Staubli VAL3: regular_pick.pgx

program regular_pick(tool x_tTool, mdesc x_mMdesc, mdesc x_mMdesc_slow, point x_pPoint_pick, dio x_dDio_cy, bool x_bBool_bk, dio x_dDio_secure)
  local point l_pPoint_pick
  local point l_pPoint_safe
  local point l_pPoint_aprch
begin

  //vertical regular pick process

  //control point preparation
  l_pPoint_safe=x_pPoint_pick
  l_pPoint_safe.trsf.z=l_pPoint_safe.trsf.z+nNum_safe_h
  //approach point preparation
  l_pPoint_aprch=x_pPoint_pick
  l_pPoint_aprch.trsf.z=l_pPoint_aprch.trsf.z+nNum_apporach_h
  //pick point preparation
  l_pPoint_pick=x_pPoint_pick

  ////to place via safe (in sequence)
  movej(l_pPoint_safe,x_tTool,x_mMdesc)
  waitEndMove()

  //corresponding cylinder extend
  if ioStatus(x_dDio_cy) >= 0
    //once io is working , on
    x_dDio_cy = true
    delay(nNum_cy_delay)
  endIf

  //open secure (on the cell not on the back secure
  if !x_bBool_bk
    call check_out_set(x_dDio_secure,true)
  endIf

  //---------------------------------
  // vertical should be linear mode
  // (Fast approach
  //---------------------------------
  movel(l_pPoint_aprch,x_tTool,x_mMdesc)
  waitEndMove()
  //---------------------------------
  // vertical should be linear mode
  // (Slow pick
  //---------------------------------
  movel(l_pPoint_pick,x_tTool,x_mMdesc_slow)
  waitEndMove()

  //vg on
  if ioStatus(x_tTool.gripper) >= 0
    //once io is working
    open(x_tTool)
  endIf

  //activate/deactive back secure if any
  if ioStatus(dDio_bk) >= 0
    //once dDio_bk is working
    dDio_bk = x_bBool_bk
    //delay to release
    delay(nNum_blow_delay)
  endIf

  //----------
  //to safe
  // (Slow up
  //----------
  movel(l_pPoint_aprch,x_tTool,x_mMdesc_slow)
  waitEndMove()
  //----------
  //to safe
  // (Fast
  //----------
  movel(l_pPoint_safe,x_tTool,x_mMdesc)
  waitEndMove()

  //corresponding cylinder extract
  if ioStatus(x_dDio_cy) >= 0
    //once io is working , off
    x_dDio_cy = false
  endIf

  //shut secure
  call check_out_set(x_dDio_secure,false)

  //check if vacuum established
  //if x_bBool_check and (dioGet(x_dDio_vs)==1)
  //success
  //elseIf x_bBool_check and (dioGet(x_dDio_vs)==1)
  //failed
  //else
  //irrelevant from IO check
  //endIf

end
